// TIA Portal V17 export
// export: Created 2025-03-05T08:01:45.6802966Z, ExportSetting WithDefaults, DisplayName Totally Integrated Automation Portal, DisplayVersion V17 Update 8, DisplayName TIA Portal Openness, DisplayVersion V17 Update 8, DisplayName TIA Portal Version Control Interface, DisplayVersion V17, DisplayName SINAMICS Startdrive Advanced, DisplayVersion V17 SP2, DisplayName SINAMICS Startdrive G110M, G120, G120C, G120D, G120P, G115D, DisplayVersion V17 SP2, DisplayName SINAMICS Startdrive G130, G150, S120, S150, SINAMICS MV, S210, DisplayVersion V17 SP2, DisplayName STEP 7 Professional, DisplayVersion V17 Update 8, DisplayName SINUMERIK ONE STEP 7 Toolbox, DisplayVersion V17 Update 12, DisplayName SINUMERIK 840D sl STEP 7 Toolbox, DisplayVersion V17 Update 12, DisplayName STEP 7 Safety, DisplayVersion V17 Update 6, DisplayName WinCC Advanced, DisplayVersion V17 Update 8
DATA_BLOCK "DB7238_HMI_WINCC_OVERVIEW"   // DB7238
{ S7_Optimized_Access := 'FALSE'; DB_Accessible_From_OPC_UA := 'FALSE' }
VERSION : 0.1
// stored: AutoNumber false, DBAccessibleFromOPCUA false, DBAccessibleFromWebserver true, IsOnlyStoredInLoadMemory false, IsWriteProtectedInAS false
   VAR
      UNIT_01_OK : Bool;   // UNIT 01 OK
      UNIT_02_OK : Bool;   // UNIT 02 OK
      U01_ASP_ALL_STA_READY : Bool;   // UNIT 01 ASPIRATION ALL STATIONS READY
      U02_ASP_ALL_STA_READY : Bool;   // UNIT 02 ASPIRATION ALL STATIONS READY
      U01_STA0_GLOBAL_ALARMS : Bool;   // UNIT 01 STATION 0 GLOBAL ALARMS
      U01_STA1_GLOBAL_ALARMS : Bool;   // UNIT 01 STATION 1 GLOBAL ALARMS
      U01_STA2_GLOBAL_ALARMS : Bool;   // UNIT 01 STATION 2 GLOBAL ALARMS
      U01_STA3_GLOBAL_ALARMS : Bool;   // UNIT 01 STATION 3 GLOBAL ALARMS
      U01_STA4_GLOBAL_ALARMS : Bool;   // UNIT 01 STATION 4 GLOBAL ALARMS
      U02_STA0_GLOBAL_ALARMS : Bool;   // UNIT 02 STATION 0 GLOBAL ALARMS
      U02_STA1_GLOBAL_ALARMS : Bool;   // UNIT 02 STATION 1 GLOBAL ALARMS
      U02_STA2_GLOBAL_ALARMS : Bool;   // UNIT 02 STATION 2 GLOBAL ALARMS
      U02_STA3_GLOBAL_ALARMS : Bool;   // UNIT 02 STATION 3 GLOBAL ALARMS
      U02_STA4_GLOBAL_ALARMS : Bool;   // UNIT 02 STATION 4 GLOBAL ALARMS
      U01_STA0_ALARMS_LED_STATUS : Int;   // UNIT 01 STATION 0 ALARMS LED STATUS
      U01_STA1_ALARMS_LED_STATUS : Int;   // UNIT 01 STATION 1 ALARMS LED STATUS
      U01_STA2_ALARMS_LED_STATUS : Int;   // UNIT 01 STATION 2 ALARMS LED STATUS
      U01_STA3_ALARMS_LED_STATUS : Int;   // UNIT 01 STATION 3 ALARMS LED STATUS
      U01_STA4_ALARMS_LED_STATUS : Int;   // UNIT 01 STATION 4 ALARMS LED STATUS
      U02_STA0_ALARMS_LED_STATUS : Int;   // UNIT 02 STATION 0 ALARMS LED STATUS
      U02_STA1_ALARMS_LED_STATUS : Int;   // UNIT 02 STATION 1 ALARMS LED STATUS
      U02_STA2_ALARMS_LED_STATUS : Int;   // UNIT 02 STATION 2 ALARMS LED STATUS
      U02_STA3_ALARMS_LED_STATUS : Int;   // UNIT 02 STATION 3 ALARMS LED STATUS
      U02_STA4_ALARMS_LED_STATUS : Int;   // UNIT 02 STATION 4 ALARMS LED STATUS
      U01_PROTEC_GAS_ALARMS_LED_STATUS : Int;   // UNIT 01 PROTECTION GAS ALARMS LED STATUS
      U02_PROTEC_GAS_ALARMS_LED_STATUS : Int;   // UNIT 02 PROTECTION GAS ALARMS LED STATUS
      U02_PROTEC_GAS_WARNINGS : Bool;   // UNIT 02 PROTECTION GAS WARNINGS
      U01_PROTEC_GAS_WARNINGS : Bool;   // UNIT 01 PROTECTION GAS WARNINGS
      COOLING_SYS_WARNINGS : Bool;   // COOLING SYSTEM WARNINGS
      COOLING_SYS_ALARMS : Bool;   // COOLING SYSTEM ALARMS
      COOLING_SYS_ALARMS_LED_STATUS : Int;   // COOLING SYSTEM ALARMS LED STATUS
      U02_ALL_ALARMS : Bool;   // UNIT 02 ALL ALARMS
      U02_ALL_WARNINGS : Bool;   // UNIT 02 ALL WARNINGS
      U02_ALL_ALARMS_LED_STATUS : Int;   // UNIT 02 ALL ALARMS LED STATUS
      U01_ALL_ALARMS : Bool;   // UNIT 01 ALL ALARMS
      U01_ALL_WARNINGS : Bool;   // UNIT 01 ALL WARNINGS
      U01_ALL_ALARMS_LED_STATUS : Int;   // UNIT 01 ALL ALARMS LED STATUS
      U01_ALL_FIXT_CLAMP_ALARMS : Bool;   // UNIT 01 ALL FIXTURES CLAMP ALARMS
      U02_ALL_FIXT_CLAMP_ALARMS : Bool;   // UNIT 02 ALL FIXTURES CLAMP ALARMS
   END_VAR
BEGIN
END_DATA_BLOCK
